PROGRAM StnBasketTotalizer
VAR

END_VAR

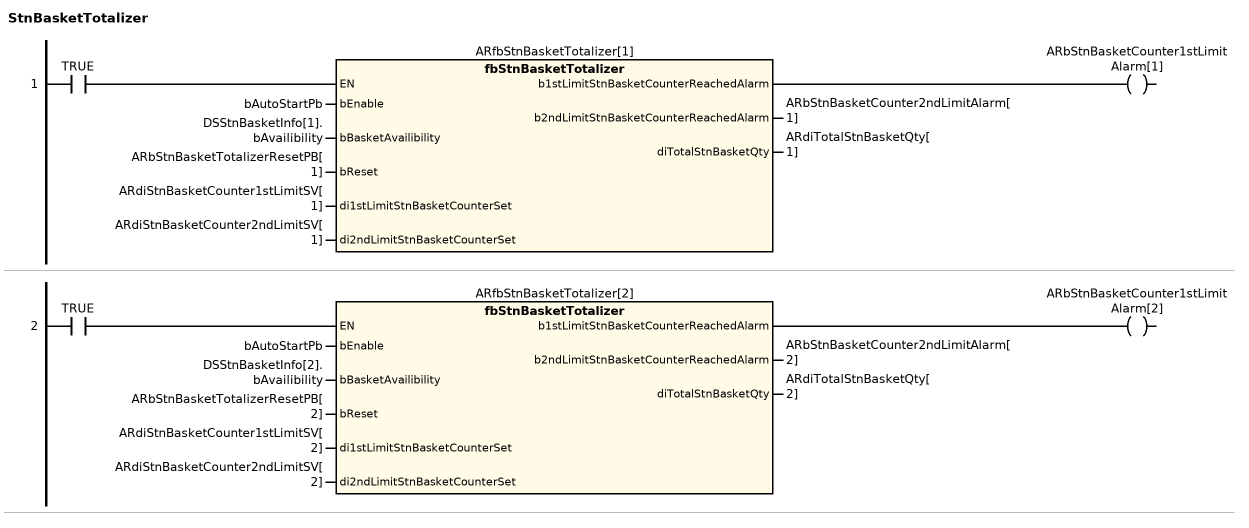
// NETWORK 1
ARfbStnBasketTotalizer[1](
    bEnable := bAutoStartPb,
    bBasketAvailibility := DSStnBasketInfo[1].bAvailibility,
    bReset := ARbStnBasketTotalizerResetPB[1],
    di1stLimitStnBasketCounterSet := ARdiStnBasketCounter1stLimitSV[1],
    di2ndLimitStnBasketCounterSet := ARdiStnBasketCounter2ndLimitSV[1],
    b2ndLimitStnBasketCounterReachedAlarm => ARbStnBasketCounter2ndLimitAlarm[1],
    diTotalStnBasketQty => ARdiTotalStnBasketQty[1]); // fbStnBasketTotalizer
ARbStnBasketCounter1stLimitAlarm[1] := ARfbStnBasketTotalizer[1].b1stLimitStnBasketCounterReachedAlarm;

// NETWORK 2
ARfbStnBasketTotalizer[2](
    bEnable := bAutoStartPb,
    bBasketAvailibility := DSStnBasketInfo[2].bAvailibility,
    bReset := ARbStnBasketTotalizerResetPB[2],
    di1stLimitStnBasketCounterSet := ARdiStnBasketCounter1stLimitSV[2],
    di2ndLimitStnBasketCounterSet := ARdiStnBasketCounter2ndLimitSV[2],
    b2ndLimitStnBasketCounterReachedAlarm => ARbStnBasketCounter2ndLimitAlarm[2],
    diTotalStnBasketQty => ARdiTotalStnBasketQty[2]); // fbStnBasketTotalizer
ARbStnBasketCounter1stLimitAlarm[2] := ARfbStnBasketTotalizer[2].b1stLimitStnBasketCounterReachedAlarm;

END_PROGRAM

(* stored: Version 1.1.0.1, ProductVersion 3.1.4024.12
   POU StnBasketTotalizer: Id {4a1b27cf-6a59-4b5d-8f6b-4025d359c190}, SpecialFunc None *)
